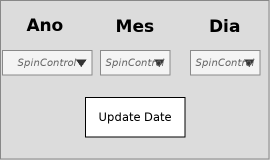
VISUALIZATION Data  // 270x160
    SpinControl (2,50 90x25), variable: GVL_TimeSch.timeToInsert.wYear
        OnMouseClick: write the text variable via Default, min 2000, max 3000
    Label (10,10 70x30), "Ano"
    SpinControl (100,50 70x25), variable: GVL_TimeSch.timeToInsert.wMonth
        OnMouseClick: write the text variable via Default, min 1, max 12
    Label (100,11 70x30), "Mes"
    SpinControl (190,50 70x25), variable: GVL_TimeSch.timeToInsert.wDay
        OnMouseClick: write the text variable via Default, min 1, max 31
    Label (190,11 70x30), "Dia"
    Rectangle (85,97 100x40), "Update Date"
        tap GVL_TimeSch.bUpdateDate
END_VISUALIZATION

(* stored: Version 1.1.0.1, ProductVersion 3.1.4024.11
   Visu Data: Id {01e19770-c16e-4399-87cd-3282732a0f30} *)
